% RSLogix 500 project CS LAB.RSS, saved by version 8.30.00.16 %
PROJECT "UNTITLED"    % processor: MicroLogix 1000 %

PROGRAM FILES
  LAD 2   7 rungs
  LAD 3, 4, 5, 6, 7, 8, 9, 10, 11, 12, 13, 14, 15, 16: only END

DATA FILES
  O0 OUTPUT  5 elements
  I1 INPUT  8 elements
  S2 STATUS  33 elements
  B3 BINARY  32 elements
  T4 TIMER  40 elements
  C5 COUNTER  32 elements
  R6 CONTROL  16 elements
  N7 INTEGER  105 elements

LADDER 2
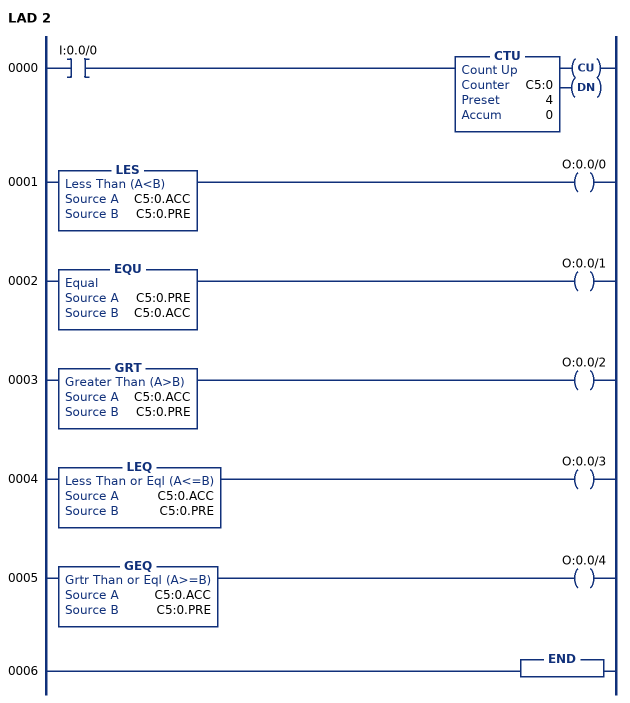
% Rung: 0 %
SOR XIC I:0.0/0 CTU C5:0 4 0 EOR
% Rung: 1 %
SOR LES C5:0.ACC C5:0.PRE OTE O:0.0/0 EOR
% Rung: 2 %
SOR EQU C5:0.PRE C5:0.ACC OTE O:0.0/1 EOR
% Rung: 3 %
SOR GRT C5:0.ACC C5:0.PRE OTE O:0.0/2 EOR
% Rung: 4 %
SOR LEQ C5:0.ACC C5:0.PRE OTE O:0.0/3 EOR
% Rung: 5 %
SOR GEQ C5:0.ACC C5:0.PRE OTE O:0.0/4 EOR
% Rung: 6 %
SOR END EOR

DATA TABLE (non-zero values as saved)
DATA C5
% .PRE .ACC %
% C5:0 % 4 0
